// SIMATIC S7-200 project (STEP 7-Micro/WIN), CPU 224 REL 02.00

ORGANIZATION_BLOCK MAIN:OB1
TITLE=PROGRAM COMMENTS
BEGIN
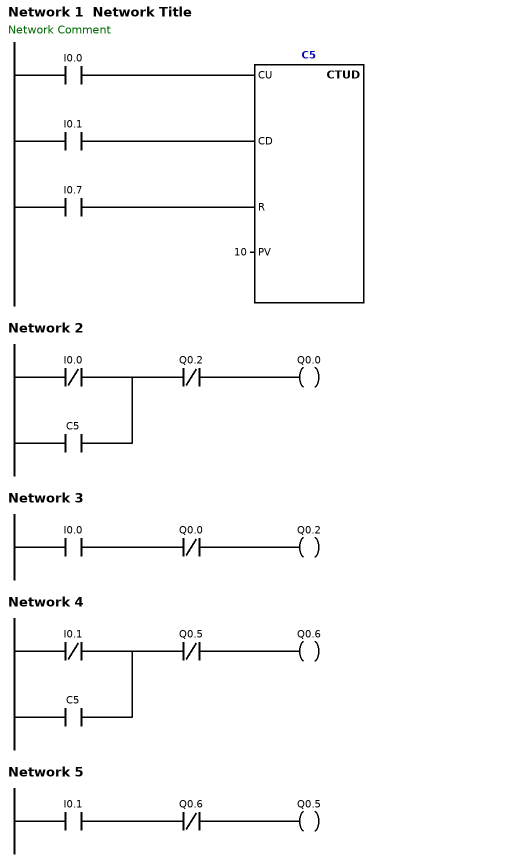
Network 1 // Network Title
// Network Comment
LD     I0.0
LD     I0.1
LD     I0.7
CTUD   C5, 10
Network 2
LDN    I0.0
O      C5
AN     Q0.2
=      Q0.0
Network 3
LD     I0.0
AN     Q0.0
=      Q0.2
Network 4
LDN    I0.1
O      C5
AN     Q0.5
=      Q0.6
Network 5
LD     I0.1
AN     Q0.6
=      Q0.5
END_ORGANIZATION_BLOCK
